// TIA Portal project "Linearachse_V16" (V16)

(* hardware
DEVICE "S71500/ET200MP-Station_1"  S7-1500 station
   slot 0: "Profilschiene_0"  Rack  6ES7 590-1***0-0AA0
   slot 1: "PLC"  CPU 1516-3 PN/DP  6ES7 516-3AN02-0AB0  V2.8
      slot 3: "CPU-Display_1"  6ES7591-1BA00-0AA0
      slot 32768: "PROFINET-Schnittstelle_1"  X1
         slot 32769: "Port_1"  X1 P1
         slot 32770: "Port_2"  X1 P2
      slot 33024: "PROFINET-Schnittstelle_2"  X2
         slot 33025: "Port_1"  X2 P1
      slot 33280: "DP-Schnittstelle_1"  X3
      slot 34817: "Virtual CP interface port_1"  Virtual CP interface port  Virtual CP interface port
*)

// ===== PLC "PLC"  CPU 1516-3 PN/DP =====

VAR_GLOBAL   // PLC tag table "Standard-Variablentabelle"
   "StörungNochNichtQuittiert" AT %M0.0 : Bool;
   "BlinkMerker" AT %M0.1 : Bool;
   "StörungAktiv" AT %M0.2 : Bool;
END_VAR

DATA_BLOCK "VersionInput"   // DB1
{ S7_Optimized_Access := 'FALSE' }
VERSION : 0.1
   VAR
      AutoTest : Bool;
      "Version" : String := 'Labor Linearantrieb V2.0';
   END_VAR
BEGIN
END_DATA_BLOCK

DATA_BLOCK "DigInput"   // DB2
{ S7_Optimized_Access := 'FALSE' }
VERSION : 0.1
   VAR
      B1 : Bool;   // Linearantrieb Endlage links → Öffner
      B2 : Bool;   // Linearantrieb Endlage rechts → Öffner
      S2 : Bool;   // Taster ( ⓪ ) → Öffner
      S1 : Bool;   // Taster ( ① ) → Schliesser
      S4 : Bool;   // Taster ( Ⅱ ) → Schliesser
      S3 : Bool;   // Taster ( Ⅰ ) → Schliesser
      S6 : Bool;   // Taster ( ↓ ) → Schliesser
      S5 : Bool;   // Taster ( ↑ ) → Schliesser
      S8 : Bool;   // Taster ( － ) → Schliesser
      S7 : Bool;   // Taster ( + ) → Schliesser
      S9 : Bool;   // Taster ( STOP ) → Öffner
      S10 : Bool;   // Not-Halt → Öffner
      S11 : Bool;   // Not-Halt → Schliesser
   END_VAR
BEGIN
END_DATA_BLOCK

DATA_BLOCK "DigOutput"   // DB3
{ S7_Optimized_Access := 'FALSE' }
VERSION : 0.1
   VAR
      Q1 : Bool;   // Linearantrieb Rechtslauf
      Q2 : Bool;   // Linearantrieb Linkslauf
      P1 : Bool;   // Meldeleuchte im Taster S1/S2 (weiß)
      P2 : Bool;   // Meldeleuchte weiß
      P3 : Bool;   // Meldeleuchte rot
      P4 : Bool;   // Meldeleuchte grün
   END_VAR
BEGIN
END_DATA_BLOCK

DATA_BLOCK "AnInput"   // DB4
{ S7_Optimized_Access := 'FALSE' }
VERSION : 0.1
BEGIN
END_DATA_BLOCK

DATA_BLOCK "AnOutput"   // DB5
{ S7_Optimized_Access := 'FALSE' }
VERSION : 0.1
BEGIN
END_DATA_BLOCK

// folder: System blocks/Program resources

DATA_BLOCK "BlinkTimer"   // DB6
{ S7_Optimized_Access := 'TRUE' }
AUTHOR : Simatic
FAMILY : IEC
NAME : IEC_TMR
VERSION : 1.0
// stored: InstanceOfName IEC_TIMER
"IEC_TIMER"
BEGIN
END_DATA_BLOCK

// folder: (top level)

FUNCTION "DatenRangieren" : Void   // FC1, SCL
{ S7_Optimized_Access := 'TRUE' }
VERSION : 0.1
   VAR_TEMP
      ErstesByte : Byte;
      ZweitesByte : Byte;
   END_VAR
BEGIN
   IF  "VersionInput".AutoTest THEN
       ; //  Es werden nur die Datenbausteine verwendet  
   ELSE
       // Digitale Eingänge I0.0 - I1.7 in den Datenbaustein DigInput DB2 kopieren
       // IB0 --> DB2 Byte 0
       // IB1 --> DB2 Byte 1
       // Area 16#81 --> Input
       // Area 16#82 --> Output
       // Area 16#84 --> DB
       #ErstesByte := PEEK(area := 16#81, dbNumber := 0, byteOffset := 0);
       #ZweitesByte := PEEK(area := 16#81, dbNumber := 0, byteOffset := 1);

       POKE(area := 16#84, dbNumber := 2, byteOffset := 0, value := #ErstesByte);
       POKE(area := 16#84, dbNumber := 2, byteOffset := 1, value := #ZweitesByte);

       // DB DigOutput auf die Ausgänge Q0.0 - Q1.7 kopieren
       // DB3 Byte 0 --> QB0
       // DB3 Byte 1 --> QB1
       #ErstesByte := PEEK(area := 16#84, dbNumber := 3, byteOffset := 0);
       #ZweitesByte := PEEK(area := 16#84, dbNumber := 3, byteOffset := 1);

       POKE(area := 16#82, dbNumber := 0, byteOffset := 0, value := #ErstesByte);
       POKE(area := 16#82, dbNumber := 0, byteOffset := 1, value := #ZweitesByte);
   END_IF;
END_FUNCTION

FUNCTION "DeleteMe" : Void   // FC2, SCL
{ S7_Optimized_Access := 'TRUE' }
VERSION : 0.1
   VAR_TEMP
      temp1 : Int;
      temp2 : Int;
   END_VAR
BEGIN
   "BlinkTimer".TON(IN := NOT "BlinkTimer".Q,
   PT := T#1250ms);

   "BlinkMerker" := "BlinkTimer".ET < T#625ms;


   IF "DigInput".S1 AND "DigInput".S2 AND NOT "StörungNochNichtQuittiert" THEN
       "DigOutput".P2 := true;
   END_IF;

   IF NOT "DigInput".S2 OR "StörungNochNichtQuittiert" THEN
       "DigOutput".P2 := FALSE;
   END_IF;

   IF NOT "DigInput".S4 OR NOT "DigInput"."S9.2" THEN
       "StörungAktiv" := true;
       "StörungNochNichtQuittiert" := true;
   END_IF;

   IF "DigInput".S4 AND "DigInput"."S9.2" THEN
       "StörungAktiv" := false;
   END_IF;

   IF (NOT "StörungAktiv" AND "DigInput".S8) THEN
       "StörungNochNichtQuittiert" := false;
   END_IF;

   "DigOutput".P3 := "StörungAktiv" OR ("StörungNochNichtQuittiert" AND "BlinkMerker");

   "DigOutput".P1 := NOT "DigOutput".P2 AND NOT "StörungNochNichtQuittiert";
END_FUNCTION

ORGANIZATION_BLOCK "Main"   // OB1, LAD, ProgramCycle
TITLE = "Main Program Sweep (Cycle)"
{ S7_Optimized_Access := 'TRUE' }
VERSION : 0.1
   VAR_INPUT
      Initial_Call : Bool;   // Initial call of this OB
      Remanence : Bool;   // =True, if remanent data are available
   END_VAR
BEGIN

REGION Network 1
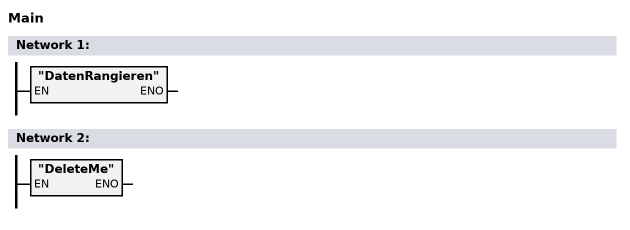
   RUNG wire#powerrail
      "DatenRangieren"()
   END_RUNG
   // the same network as SCL:
   "DatenRangieren"();
END_REGION

REGION Network 2
   RUNG wire#powerrail
      "DeleteMe"()
   END_RUNG
   // the same network as SCL:
   "DeleteMe"();
END_REGION
END_ORGANIZATION_BLOCK

ORGANIZATION_BLOCK "Startup"   // OB100, SCL, Startup
TITLE = "Complete Restart"
{ S7_Optimized_Access := 'TRUE' }
VERSION : 0.1
   VAR_INPUT
      LostRetentive : Bool;   // True if retentive data are lost
      LostRTC : Bool;   // True if date and time are lost
   END_VAR
BEGIN
   POKE(area := 16#84,     // DB
        dbNumber := 3,     // DB DigOutput
        byteOffset := 0,   // Byte 0
        value := byte#0);  // löschen

   POKE(area := 16#84,     // DB
        dbNumber := 3,     // DB Digoutput
        byteOffset := 1,   // Byte 1
        value := byte#0);  // löschen
END_ORGANIZATION_BLOCK